FUNCTION_BLOCK FB_Cylinder
VAR_INPUT
END_VAR
VAR_OUTPUT
END_VAR
VAR
	bExtended		: BOOL;
	bExtendCmd		: BOOL;
	bRetractCmd		: BOOL;
	
	sName			: STRING;
	ton				: TON;
	nState			: DINT;
END_VAR

PROPERTY Extended : BOOL
GET
Extended := bExtended;
END_GET
SET
bExtended := Extended;
END_SET
END_PROPERTY

METHOD Manual : BOOL
VAR_INPUT
END_VAR
CASE nState OF
	0:
		bExtended := FALSE;
		IF bExtendCmd THEN
			ton(IN:=TRUE, PT:=T#1S);
			IF ton.Q THEN
				nState := 1;
			END_IF
		END_IF
	1:
		bExtended := TRUE;
		IF bRetractCmd THEN
			ton(IN:=FALSE);
			nState := 0;
		END_IF
END_CASE
END_METHOD

PROPERTY Name : STRING
GET
Name := sName;
END_GET
SET
sName := Name;
END_SET
END_PROPERTY

END_FUNCTION_BLOCK

(* stored: Version 1.1.0.1
   POU FB_Cylinder: Id {91e06a43-077e-41ea-99f6-fff253614575}, SpecialFunc None
   Property Extended: Id {b8001383-c48e-43ac-b7e5-f8de451ae12e}
   Get Get: Id {3e9e7f51-d230-412b-9827-30de6f4413b2}
   Set Set: Id {a74159aa-2143-4eb5-ad83-52d8fb65b319}
   Method Manual: Id {1719d544-aee5-42b7-b3f8-e15f21ac5362}
   Property Name: Id {2f360821-dde2-4298-a722-1154d6811004}
   Get Get: Id {e35b105e-4f19-43ac-be2f-0a5250439b38}
   Set Set: Id {c548a2b7-0ad9-4628-bcdf-8afa00dc309a} *)
